(* PLC project Sin nombre, Desconocido Sin nombre 1 *)
(* stored: creationDateTime 2023-10-03T11:15:35, modificationDateTime 2023-10-03T12:08:24 *)

PROGRAM exam_openPLC_simu
  VAR
    s1_arrive AT %IX0.0 : BOOL;  (* IN_bottle arrives to be filled *)
    s2_arrive AT %IX0.1 : BOOL;  (* IN_bottle arrives to be sealed *)
    s3_bottle_full AT %IX0.2 : BOOL;  (* IN_bottle is full? *)
    s4_bottle_seal AT %IX0.3 : BOOL;  (* IN_bottle was sealed? *)
    start AT %IX0.4 : BOOL;  (* IN_start proccess *)
    bomb AT %QX0.0 : BOOL;  (* OUT_bomb is active? *)
    Ms_down_up AT %QX0.1 : BOOL;  (* OUT_seal is active *)
    M1_M2 AT %QX0.2 : BOOL;  (* OUT_band is active *)
  END_VAR
  VAR
    TON0 : TON;  (* sealing time *)
  END_VAR

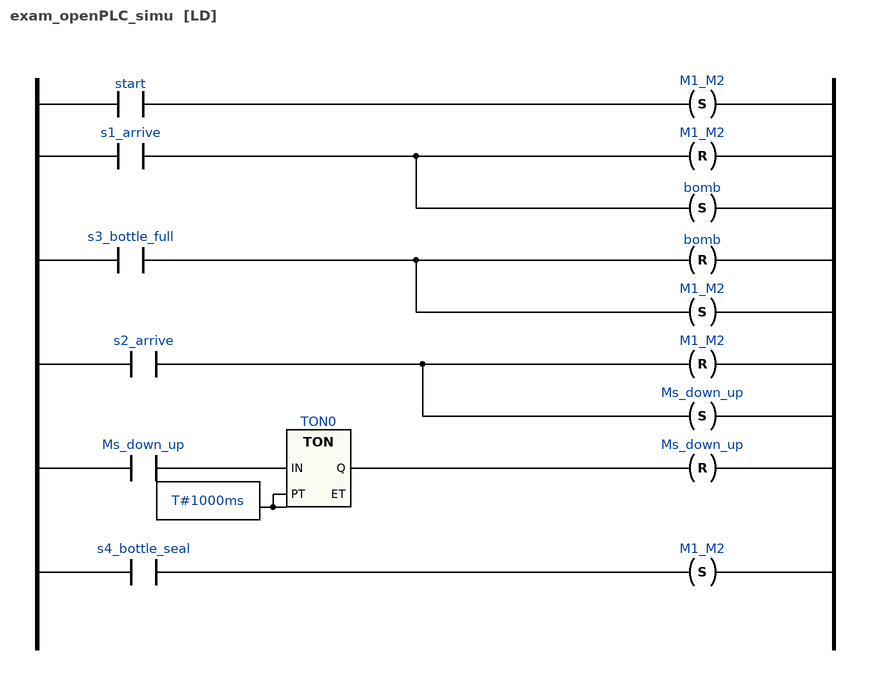
(* LD diagram, written out as Structured Text *)
IF start THEN M1_M2 := TRUE; END_IF;
IF s1_arrive THEN M1_M2 := FALSE; END_IF;
IF s1_arrive THEN bomb := TRUE; END_IF;
IF s3_bottle_full THEN bomb := FALSE; END_IF;
IF s3_bottle_full THEN M1_M2 := TRUE; END_IF;
IF s2_arrive THEN M1_M2 := FALSE; END_IF;
IF s2_arrive THEN Ms_down_up := TRUE; END_IF;
TON0(IN := Ms_down_up, PT := T#1000ms);
IF TON0.Q THEN Ms_down_up := FALSE; END_IF;
IF s4_bottle_seal THEN M1_M2 := TRUE; END_IF;
END_PROGRAM

CONFIGURATION Config0
  RESOURCE Res0 ON PLC
    TASK task0(INTERVAL := T#20ms, PRIORITY := 0);
    PROGRAM instance0 WITH task0 : exam_openPLC_simu;
  END_RESOURCE
END_CONFIGURATION
